// TwinCAT 3 PLC project PLC
// ProgramVersion: 3.1.4024.0
// libraries:
//   Tc2_Standard, * (Beckhoff Automation GmbH)
//   Tc2_System, * (Beckhoff Automation GmbH)
//   Tc3_Module, * (Beckhoff Automation GmbH)
//   VisuSymbols,3.5.10.0,System
// project tree:
//   DUTs/ stShiftRegData.TcDUT
//   / GlobalTextList.TcGTLO, PlcTask.TcTTO
//   POUs/FB/ ConveyorTracking.TcPOU, Fifo.TcPOU, ShiftRegister.TcPOU
//   POUs/ MAIN.TcPOU
//   Simulation/ DriveSimulator.TcPOU, Simulation.TcPOU
//   VISUs/ Visualization.TcVIS, VisualizationManager.TcVMO (not stored)
// real-time tasks:
//   TASK PlcTask: cycle T#10ms, priority 20, ADS port 350

CONFIGURATION PLC
    RESOURCE PLC ON TwinCAT3
        TASK PlcTask(INTERVAL := T#10ms, PRIORITY := 20);
        PROGRAM MAIN WITH PlcTask : MAIN;
    END_RESOURCE
END_CONFIGURATION

// ---- DUTs/stShiftRegData.TcDUT
(*Shift Register Data Structure*)
TYPE stShiftRegData :
STRUCT
	ProductSts	:	BOOL;			// True=product present
	ProductType	:	INT:=-1;		// 1=big product; 2=middle product; 3=small product
END_STRUCT
END_TYPE

// ---- POUs/MAIN.TcPOU
PROGRAM MAIN
VAR
	ConveyorTracking01		: 	ConveyorTracking;	
	ConveyorTracking02		: 	ConveyorTracking;
	ConveyorTracking03		: 	ConveyorTracking;
	EncoderResolution		:	REAL:=0.2;
	TrackingAccuracy		:	REAL:=1.0;
	Reset					: 	BOOL;
	tpDrvStop				: 	TP;
	DroppedProducts1		:	CTU;
	DroppedProducts2		:	CTU;
	DroppedProducts3		:	CTU;
END_VAR

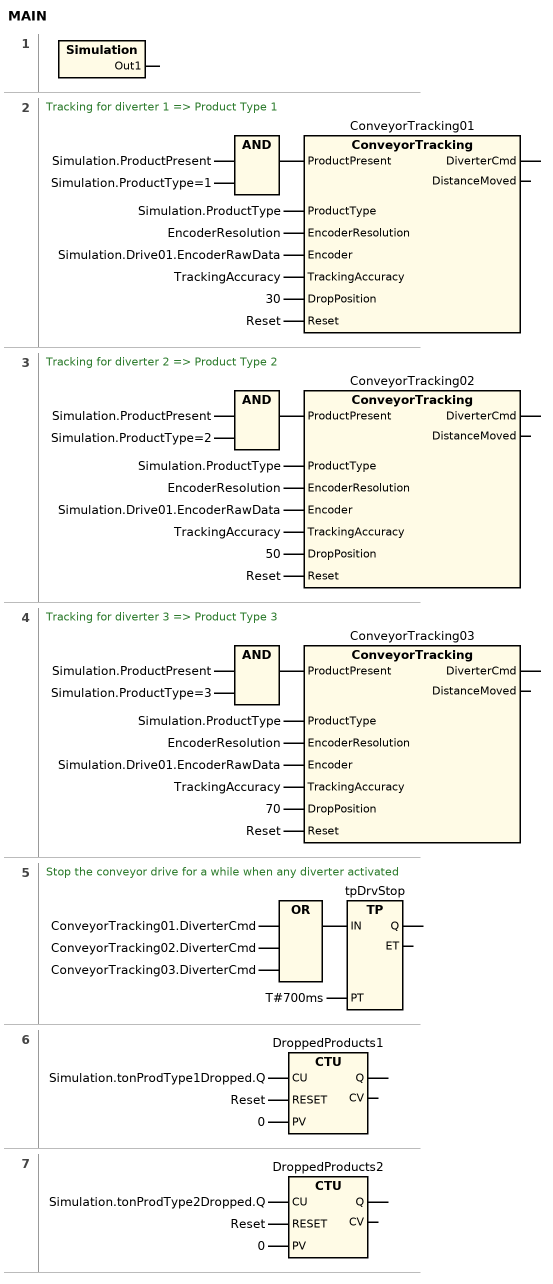
// NETWORK 1
Simulation();

// NETWORK 2
// Tracking for diverter 1 => Product Type 1
ConveyorTracking01(
    ProductPresent := Simulation.ProductPresent AND (Simulation.ProductType=1),
    ProductType := Simulation.ProductType,
    EncoderResolution := EncoderResolution,
    Encoder := Simulation.Drive01.EncoderRawData,
    TrackingAccuracy := TrackingAccuracy,
    DropPosition := 30,
    Reset := Reset); // ConveyorTracking

// NETWORK 3
// Tracking for diverter 2 => Product Type 2
ConveyorTracking02(
    ProductPresent := Simulation.ProductPresent AND (Simulation.ProductType=2),
    ProductType := Simulation.ProductType,
    EncoderResolution := EncoderResolution,
    Encoder := Simulation.Drive01.EncoderRawData,
    TrackingAccuracy := TrackingAccuracy,
    DropPosition := 50,
    Reset := Reset); // ConveyorTracking

// NETWORK 4
// Tracking for diverter 3 => Product Type 3
ConveyorTracking03(
    ProductPresent := Simulation.ProductPresent AND (Simulation.ProductType=3),
    ProductType := Simulation.ProductType,
    EncoderResolution := EncoderResolution,
    Encoder := Simulation.Drive01.EncoderRawData,
    TrackingAccuracy := TrackingAccuracy,
    DropPosition := 70,
    Reset := Reset); // ConveyorTracking

// NETWORK 5
// Stop the conveyor drive for a while when any diverter activated
tpDrvStop(IN := ConveyorTracking01.DiverterCmd OR ConveyorTracking02.DiverterCmd OR ConveyorTracking03.DiverterCmd, PT := T#700ms); // TP

// NETWORK 6
DroppedProducts1(CU := Simulation.tonProdType1Dropped.Q, RESET := Reset, PV := 0); // CTU

// NETWORK 7
DroppedProducts2(CU := Simulation.tonProdType2Dropped.Q, RESET := Reset, PV := 0); // CTU

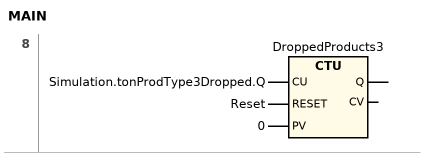
// NETWORK 8
DroppedProducts3(CU := Simulation.tonProdType3Dropped.Q, RESET := Reset, PV := 0); // CTU

END_PROGRAM

// ---- POUs/FB/ConveyorTracking.TcPOU
FUNCTION_BLOCK ConveyorTracking
VAR_INPUT
	ProductPresent				:	BOOL;		// sensor detecting the product at the start of the conveyor
	ProductType					:	INT;		// product type
	EncoderResolution			:	REAL;		// how many mm distance per one encoder pulse [mm/pulses]
	Encoder						:	LINT;		// raw encoder value in pulses	
	TrackingAccuracy			:	REAL;		// needed product tracking accuracy [mm]
	DropPosition				:	UINT;		// diverter position in [mm]

	Reset						:	BOOL;		// reset all tracking logic
END_VAR
VAR_OUTPUT
	DiverterCmd					:	BOOL;		// command to activate the diverter
	DistanceMoved				:	REAL;		// distance a product has moved since product presence sensor
END_VAR
VAR
	Init						:	BOOL:=TRUE;
	EncValueMem					:	LINT;
	EncDiff						: 	LINT;
	
	rtTrack						: 	R_TRIG;
	TrackTrigger				: 	BOOL;
	
	Register					:	ARRAY[0..500] OF stShiftRegData;
	ShiftRegister01				: 	ShiftRegister;
	ctuProductLen				: 	CTU;
	ftrigProduct				: 	F_TRIG;
	ProductLen					:	WORD;
	FifoLoad					: 	Fifo;
	MiddlePointPos				: 	REAL;

	rtrigProductPresent			: 	R_TRIG;
	ProductStarted				: 	BOOL;
	ftrigProductGone			: 	F_TRIG;
END_VAR
VAR // added by the converter: edge detectors and wires of the graphical bodies
    _w1, _w2 : BOOL;
END_VAR

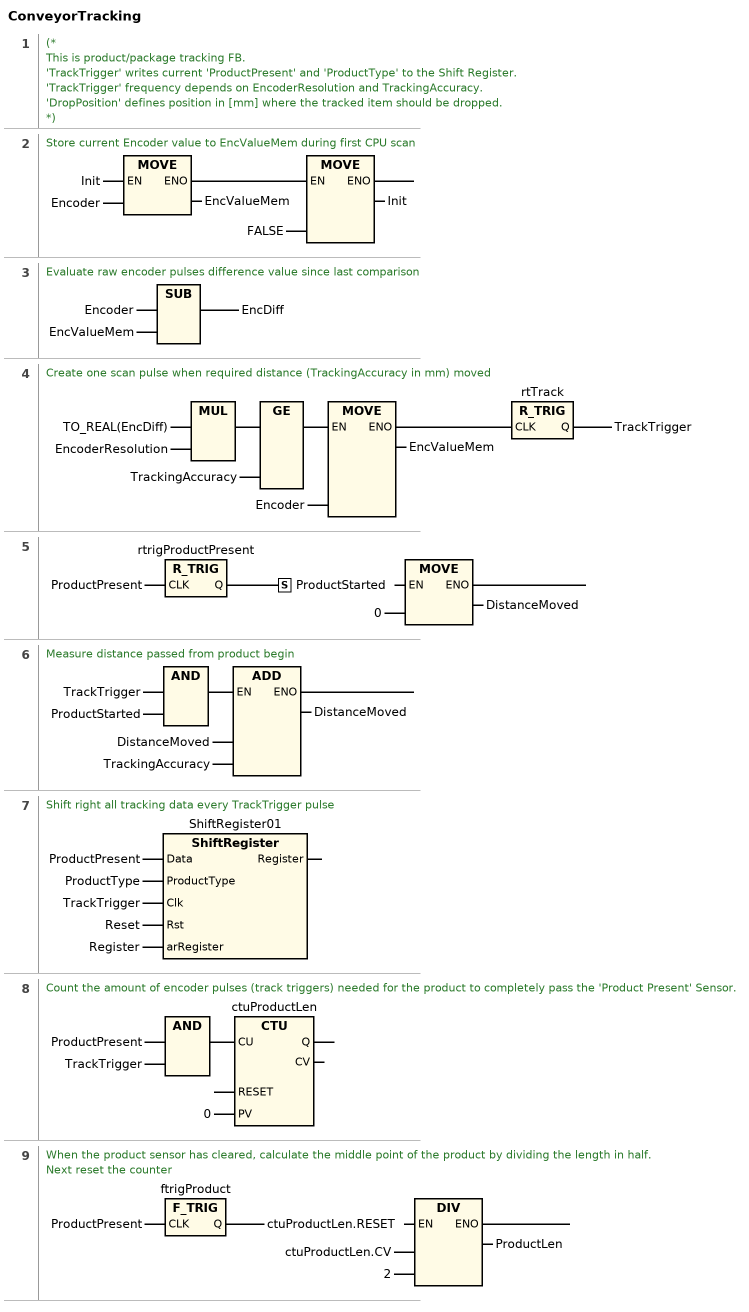
// NETWORK 1
// (*
// This is product/package tracking FB.
// 'TrackTrigger' writes current 'ProductPresent' and 'ProductType' to the Shift Register.
// 'TrackTrigger' frequency depends on EncoderResolution and TrackingAccuracy.
// 'DropPosition' defines position in [mm] where the tracked item should be dropped.
// *)

// NETWORK 2
// Store current Encoder value to EncValueMem during first CPU scan
_w1 := Init;
IF _w1 THEN EncValueMem := Encoder; END_IF
IF _w1 THEN Init := FALSE; END_IF

// NETWORK 3
// Evaluate raw encoder pulses difference value since last comparison
EncDiff := Encoder - EncValueMem;

// NETWORK 4
// Create one scan pulse when required distance (TrackingAccuracy in mm) moved
_w2 := (TO_REAL(EncDiff)) * EncoderResolution >= TrackingAccuracy;
IF _w2 THEN EncValueMem := Encoder; END_IF
rtTrack(CLK := _w2); // R_TRIG
TrackTrigger := rtTrack.Q;

// NETWORK 5
rtrigProductPresent(CLK := ProductPresent); // R_TRIG
ProductStarted S= rtrigProductPresent.Q;
IF rtrigProductPresent.Q THEN DistanceMoved := 0; END_IF

// NETWORK 6
// Measure distance passed from product begin
IF TrackTrigger AND ProductStarted THEN DistanceMoved := DistanceMoved + TrackingAccuracy; END_IF

// NETWORK 7
// Shift right all tracking data every TrackTrigger pulse
ShiftRegister01(
    Data := ProductPresent,
    ProductType := ProductType,
    Clk := TrackTrigger,
    Rst := Reset,
    arRegister := Register); // ShiftRegister

// NETWORK 8
// Count the amount of encoder pulses (track triggers) needed for the product to completely pass the 'Product Present' Sensor.
ctuProductLen(CU := ProductPresent AND TrackTrigger, PV := 0); // CTU

// NETWORK 9
// When the product sensor has cleared, calculate the middle point of the product by dividing the length in half.
// Next reset the counter
ftrigProduct(CLK := ProductPresent); // F_TRIG
ctuProductLen.RESET := ftrigProduct.Q;
IF ftrigProduct.Q THEN ProductLen := ctuProductLen.CV / 2; END_IF

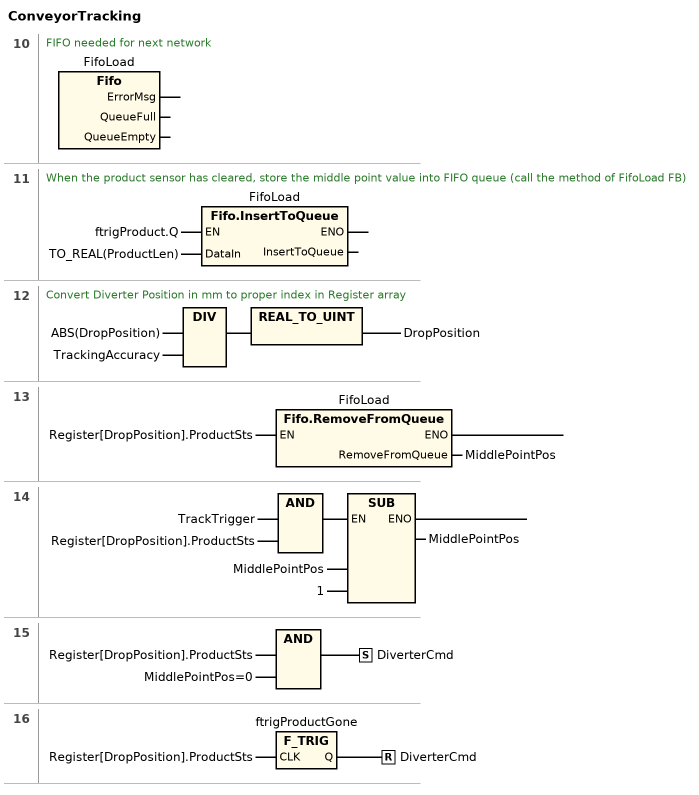
// NETWORK 10
// FIFO needed for next network
FifoLoad(); // Fifo

// NETWORK 11
// When the product sensor has cleared, store the middle point value into FIFO queue (call the method of FifoLoad FB)
IF ftrigProduct.Q THEN FifoLoad.InsertToQueue(DataIn := TO_REAL(ProductLen)); END_IF

// NETWORK 12
// Convert Diverter Position in mm to proper index in Register array
DropPosition := REAL_TO_UINT((ABS(DropPosition)) / TrackingAccuracy);

// NETWORK 13
IF Register[DropPosition].ProductSts THEN FifoLoad.RemoveFromQueue(RemoveFromQueue => MiddlePointPos); END_IF

// NETWORK 14
IF TrackTrigger AND Register[DropPosition].ProductSts THEN MiddlePointPos := MiddlePointPos - 1; END_IF

// NETWORK 15
DiverterCmd S= Register[DropPosition].ProductSts AND (MiddlePointPos=0);

// NETWORK 16
ftrigProductGone(CLK := Register[DropPosition].ProductSts); // F_TRIG
DiverterCmd R= ftrigProductGone.Q;

END_FUNCTION_BLOCK

// ---- POUs/FB/ShiftRegister.TcPOU
FUNCTION_BLOCK ShiftRegister
VAR_INPUT
	Data			: 	BOOL;
	ProductType		:	INT;
	Clk				: 	BOOL;
	Rst				: 	BOOL;
END_VAR

VAR
	rtrigClk 		: 	R_TRIG;
	Idx				:	UINT;
END_VAR

VAR_IN_OUT
	arRegister			:	ARRAY[0..500] OF stShiftRegData;
END_VAR

VAR_OUTPUT

END_VAR

(*
Shift register for complex(STRUCT) data type

Each CLK signal stores 'Data' and 'ProductType'
into first position of the register as STRUCT data type.
All other entries from the register will be then shifted by one position. 
*)

// detect rising edge on clk signal
rtrigClk(clk := Clk);

IF rtrigClk.Q THEN
	FOR Idx := 500 TO 1 BY -1 DO
		arRegister[Idx] := arRegister[Idx-1];
	END_FOR
	arRegister[0].ProductSts := Data;
	arRegister[0].ProductType := ProductType;
	
END_IF

IF Rst THEN
	MEMSET(ADR(arRegister), 0, SIZEOF(arRegister) );
END_IF

END_FUNCTION_BLOCK

// ---- POUs/FB/Fifo.TcPOU
FUNCTION_BLOCK Fifo

VAR_OUTPUT
	ErrorMsg			:	STRING(50);	// error message
	QueueFull			:	Bool;
	QueueEmpty			:	BOOL;
END_VAR

VAR CONSTANT
	QueueMin			: 	INT:=0;
	QueueMax			:	INT:=29;
END_VAR

VAR
	ptrHead				:	INT ;		// pointer to first element (head)
	ptrTail				:	INT ; 		// pointer to last element (tail) 
	Idx					:	INT;
	InitBit				:	BOOL:=TRUE;
	QueueSize			:	INT;		// size of circular queue
	QueueSizeOk			:	BOOL;		
	Queue				:	ARRAY[QueueMin..QueueMax] OF REAL;
	// test:
	QueueLength			:	INT:=8;
END_VAR

(*
This FB acts as FIFO i.e. circular queue.
Size of the queue must be customized with constants QueueMin and QueueMax. 
*)
IF InitBit THEN

	InitBit := FALSE;
	
	IF QueueMax > QueueMin THEN
		ptrHead := -1;
		ptrTail := -1;
		QueueSize := TO_INT(SIZEOF(Queue) / SIZEOF(REAL));
		QueueSizeOk := TRUE;
	END_IF
END_IF

METHOD ClearQueue : BOOL
VAR_INPUT
END_VAR
(* reinit the queue *)

IF QueueSizeOk THEN
	ptrHead := -1;
	ptrTail := -1;
	
	FOR Idx := QueueMin TO QueueMax DO
		Queue[Idx] := 0;
	END_FOR

	ErrorMsg := '';
	QueueEmpty := FALSE;
	QueueFull := FALSE;
END_IF
END_METHOD

METHOD InsertToQueue : BOOL
VAR_INPUT
	DataIn		:	REAL;			// data to insert into circular queue
END_VAR
// Insert new data into queue

IF QueueSizeOk THEN 
	IF IsFull THEN
		// queue is full. can't insert new data
		ErrorMsg := 'Queue is full. Can not insert new data';
		QueueFull := TRUE;
	ELSIF IsEmpty THEN
		ErrorMsg := '';
		QueueFull := FALSE;
		ptrHead := 0;
		ptrTail := 0;
		Queue[ptrTail] := DataIn;
	ELSE 
		ErrorMsg := '';
		QueueFull := FALSE;
		IF (ptrTail+1) MOD QueueLength <= QueueLength THEN
			ptrTail := (ptrTail + 1) MOD QueueLength;
			Queue[ptrTail] := DataIn;	
		END_IF
	
	END_IF
END_IF
END_METHOD

PROPERTY IsEmpty : BOOL
GET
IsEmpty := ptrHead = -1 AND ptrTail = -1;
END_GET
END_PROPERTY

PROPERTY IsFull : BOOL
GET
IsFull := ptrHead = (ptrTail + 1) MOD QueueLength;
END_GET
END_PROPERTY

PROPERTY NoOfDataPoints : INT
GET
// number of data points in queue
IF ptrTail>ptrHead THEN
	NoOfDataPoints:=ABS(ptrTail - ptrHead)+1;
ELSIF ptrTail<ptrHead THEN
	NoOfDataPoints:=(ptrTail+1) + (QueueLength-ptrHead);
ELSE
	// ptrTail=ptrHead
	NoOfDataPoints:=0;
END_IF
END_GET
END_PROPERTY

METHOD RemoveFromQueue : Real;
VAR_INPUT
END_VAR
(* remove one data from the queue *)

IF QueueSizeOk THEN
	IF IsEmpty THEN							// zero element in queue
		ErrorMsg := 'Queue is empty';
		QueueEmpty := TRUE;
	ELSIF ptrHead=ptrTail THEN				// only one element in queue
		ErrorMsg := '';
		QueueEmpty := FALSE;
		RemoveFromQueue := Queue[ptrHead];
		Queue[ptrHead]:=0;
		ptrHead := -1;
		ptrTail := -1;
	ELSE									// more then one element in queue
		ErrorMsg := '';
		QueueEmpty := FALSE;
		IF (ptrHead + 1) MOD QueueLength <= QueueLength THEN
			RemoveFromQueue := Queue[ptrHead];
			Queue[ptrHead]:=0;
			ptrHead := (ptrHead + 1) MOD QueueLength;
		END_IF
	END_IF
END_IF
END_METHOD

END_FUNCTION_BLOCK

// ---- Simulation/Simulation.TcPOU
PROGRAM Simulation
VAR
	Drive01			:	DriveSimulator;
	CmdDrv01		:	BOOL;
	ProductPresent	:	BOOL;
	ProductType		:	INT;
	RndGen			:	Drand;
	RndNum			:	LREAL;
	tp01			:	TP;
	tp02			:	TP;
	rtrig01			:	R_TRIG;
	tpProductTypeRead	:	TP;

	tonProdType1Dropped: TON;
	tonProdType2Dropped: TON;
	tonProdType3Dropped: TON;
END_VAR

// simulate conveyor drive
Drive01(CmdRun:=CmdDrv01 AND NOT Main.tpDrvStop.Q , EncoderRawData=> );

// pulse generation for product availability 
IF Drive01.DrvRunning THEN
	tp01(IN:=NOT tp02.Q , PT:=T#15S , Q=> , ET=> );
	tp02(IN:=NOT tp01.Q , PT:=T#1.5S , Q=> , ET=> );
	rtrig01(CLK:=tp02.Q);
ELSE
	tp01(IN:=FALSE);
	tp02(IN:=FALSE);
END_IF;

//simulate product type reader
tpProductTypeRead(IN:=rtrig01.Q, PT:=T#600MS);

// simulate frequently product generation when drive is running
IF Drive01.DrvRunning  AND rtrig01.Q THEN	
	RndGen(Seed:=2);
	RndNum := RndGen.Num;
	IF RndNum < 0.5 THEN
		ProductType := 1;
	ELSIF RndNum < 0.8 THEN
		ProductType := 2;
	ELSE
		ProductType := 3;
	END_IF
	
END_IF

// simulate product presence and product type during pulse=TRUE
ProductPresent := Drive01.DrvRunning AND tp02.Q;


// simulate sensors for dropping products
tonProdType1Dropped(IN:=MAIN.ConveyorTracking01.DiverterCmd, 
					PT:=T#700MS, 
					Q=>, 
					ET=> );

tonProdType2Dropped(IN:=MAIN.ConveyorTracking02.DiverterCmd, 
					PT:=T#700MS, 
					Q=>, 
					ET=> );
					
tonProdType3Dropped(IN:=MAIN.ConveyorTracking03.DiverterCmd, 
					PT:=T#700MS, 
					Q=>, 
					ET=> );

END_PROGRAM

// ---- Simulation/DriveSimulator.TcPOU
FUNCTION_BLOCK DriveSimulator
VAR_INPUT
	CmdRun			:	BOOL;
END_VAR
VAR_OUTPUT
	DrvRunning		:	BOOL;
	EncoderRawData	:	LINT;
END_VAR
VAR
	tp01			: TP;
	tp02			: TP;
	rtrig01			: R_TRIG;
END_VAR

(*
FB simulates conveyor motor with position encoder
Inputs:
	CmdRun:	start drive to run
Outputs:
	DrvRunning:	status for drive running
	EncoderRawData: encoder position
*)
IF CmdRun THEN
	DrvRunning := TRUE;
	tp01(IN:=NOT tp02.Q , PT:=T#10MS , Q=> , ET=> );
	tp02(IN:=NOT tp01.Q , PT:=T#10MS , Q=> , ET=> );
	rtrig01(CLK:=tp02.Q);
	
	IF rtrig01.Q THEN
		EncoderRawData :=  EncoderRawData + 1;
	END_IF
ELSE
	DrvRunning := FALSE;
END_IF

END_FUNCTION_BLOCK

// ---- GlobalTextList.TcGTLO
TEXTLIST GlobalTextList
  225 = '1'
  361 = '2'
  150 = '3'
  329 = 'Motor'
  271 = 'Product Tracking'
  738 = 'Product Type 1 \nAmount: \n%s'
  750 = 'Product Type 2\nAmount: \n%s'
  344 = 'Product Type 3 \nAmount: \n%s'
  396 = 'Product Type Reader'
  544 = 'RESET'
  814 = 'RUN'
END_TEXTLIST

// ---- VISUs/Visualization.TcVIS
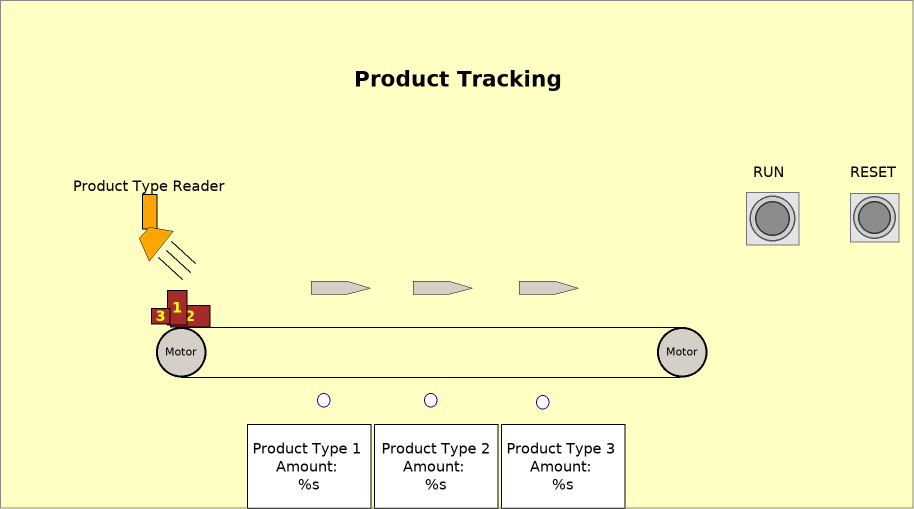
VISUALIZATION Visualization  // 914x509
    PushSwitchLed (746,191 53x55), variable: Simulation.CmdDrv01, behaviour: TOGGLE, style: Switch-PushSwitchLed-Gray
    Ellipse (156,327 50x50), "Motor", colour toggle: Simulation.Drive01.DrvRunning
    Label (728,157 82x30), "RUN"
    Label (832,157 82x30), "RESET"
    Ellipse (657,327 50x50), "Motor", colour toggle: Simulation.Drive01.DrvRunning
    Line (183,327) (680,327)
    Rectangle (142,194 15x35), angle 310
    Label (64,171 170x30), "Product Type Reader"
    Line (181,377) (680,377)
    Polygon (311,281) (347,281) (370,288) (347,294) (311,294)
        p2858320360: BOOL_TO_INT(MAIN.ConveyorTracking01.DiverterCmd) * 90
    Polygon (413,281) (449,281) (472,288) (449,294) (413,294)
        p2858320360: BOOL_TO_INT(MAIN.ConveyorTracking02.DiverterCmd) * 90
    Polygon (519,281) (555,281) (578,288) (555,294) (519,294)
        p2858320360: BOOL_TO_INT(MAIN.ConveyorTracking03.DiverterCmd) * 90
    Rectangle (170,305 40x22), "2", invisible if: Simulation.ProductType <> 2 OR MAIN.ConveyorTracking02.DistanceMoved > 52
        p3560616238: MAIN.ConveyorTracking02.DistanceMoved * 3.9
    Rectangle (167,290 20x35), "1", invisible if: Simulation.ProductType <> 1 OR MAIN.ConveyorTracking01.DistanceMoved > 32
        p3560616238: MAIN.ConveyorTracking01.DistanceMoved * 4.0
    Rectangle (151,308 19x16), "3", invisible if: Simulation.ProductType <> 3 OR MAIN.ConveyorTracking03.DistanceMoved > 72
        p3560616238: MAIN.ConveyorTracking03.DistanceMoved * 4.8
    Rectangle (247,424 124x85), "Product Type 1 Amount: %s", text variable: MAIN.DroppedProducts1.CV
    Ellipse (317,393 13x14), colour toggle: Simulation.tonProdType1Dropped.Q
    Ellipse (424,393 13x14), colour toggle: Simulation.tonProdType2Dropped.Q
    Ellipse (536,395 13x14), colour toggle: Simulation.tonProdType3Dropped.Q
    PushSwitch (850,191 49x53), variable: MAIN.Reset, behaviour: TAP, style: Switch-PushSwitch-Gray
    Rectangle (374,424 124x85), "Product Type 2 Amount: %s", text variable: MAIN.DroppedProducts2.CV
    Rectangle (501,424 124x85), "Product Type 3 Amount: %s", text variable: MAIN.DroppedProducts3.CV
    Label (322,64 272x30), "Product Tracking"
    Polygon (139,238) (149,227) (173,231) (149,261), colour toggle: Simulation.tpProductTypeRead.Q
    Line (171,241) (195,263), invisible if: NOT Simulation.tpProductTypeRead.Q
        p2086823670: NOT Simulation.tpProductTypeRead.Q
    Line (166,250) (190,272), invisible if: NOT Simulation.tpProductTypeRead.Q
        p2086823670: NOT Simulation.tpProductTypeRead.Q
    Line (158,257) (182,279), invisible if: NOT Simulation.tpProductTypeRead.Q
        p2086823670: NOT Simulation.tpProductTypeRead.Q
END_VISUALIZATION
